// TIA Portal V17 export
// export: Created 2024-08-26T21:07:22.3455674Z, ExportSetting WithDefaults, DisplayName Totally Integrated Automation Portal, DisplayVersion V17 Update 7, DisplayName TIA Portal Openness, DisplayVersion V17 Update 7, DisplayName TIA Portal Version Control Interface, DisplayVersion V17, DisplayName SINAMICS Startdrive Advanced, DisplayVersion V17 SP2, DisplayName SINAMICS Startdrive G110M, G120, G120C, G120D, G120P, G115D, DisplayVersion V17 SP2, DisplayName SINAMICS Startdrive G130, G150, S120, S150, SINAMICS MV, S210, DisplayVersion V17 SP2, DisplayName STEP 7 Professional, DisplayVersion V17 Update 7, DisplayName STEP 7 Safety, DisplayVersion V17 Update 6, DisplayName WinCC Advanced / Unified PC, DisplayVersion V17 Update 7
VAR_GLOBAL   // PLC tag table "codeReaderMemory"
   reqScannerConfig AT %M2250.2 : Bool;
   bufferReset AT %M2250.0 : Bool;
   labelReadingError AT %M186.3 : Bool;
   labelNok AT %M187.0 : Bool;
   nestLabelReadingError AT %M224.0 : Bool;
   idleTime AT %M2250.1 : Bool;
   seatLabelIdentified AT %M2250.3 : Bool;
   motorLabelIdentified AT %M2250.4 : Bool;
   xLabelIdentified AT %M2250.5 : Bool;
   hmiNestScannerReq AT %M2.3 : Bool;
   scannerOnConfig AT %M2.6 : Bool;
   scanningNest AT %M2.7 : Bool;
   nestCodeRead AT %M3.3 : Bool;
   upperScannerCodeRead AT %M3.4 : Bool;
   angleScannerCodeRead AT %M3.7 : Bool;
   scanningAngle AT %M4.2 : Bool;
   scanningUpper AT %M4.6 : Bool;
   label1Upper AT %M8.2 : Bool;
   label2Upper AT %M8.3 : Bool;
END_VAR
